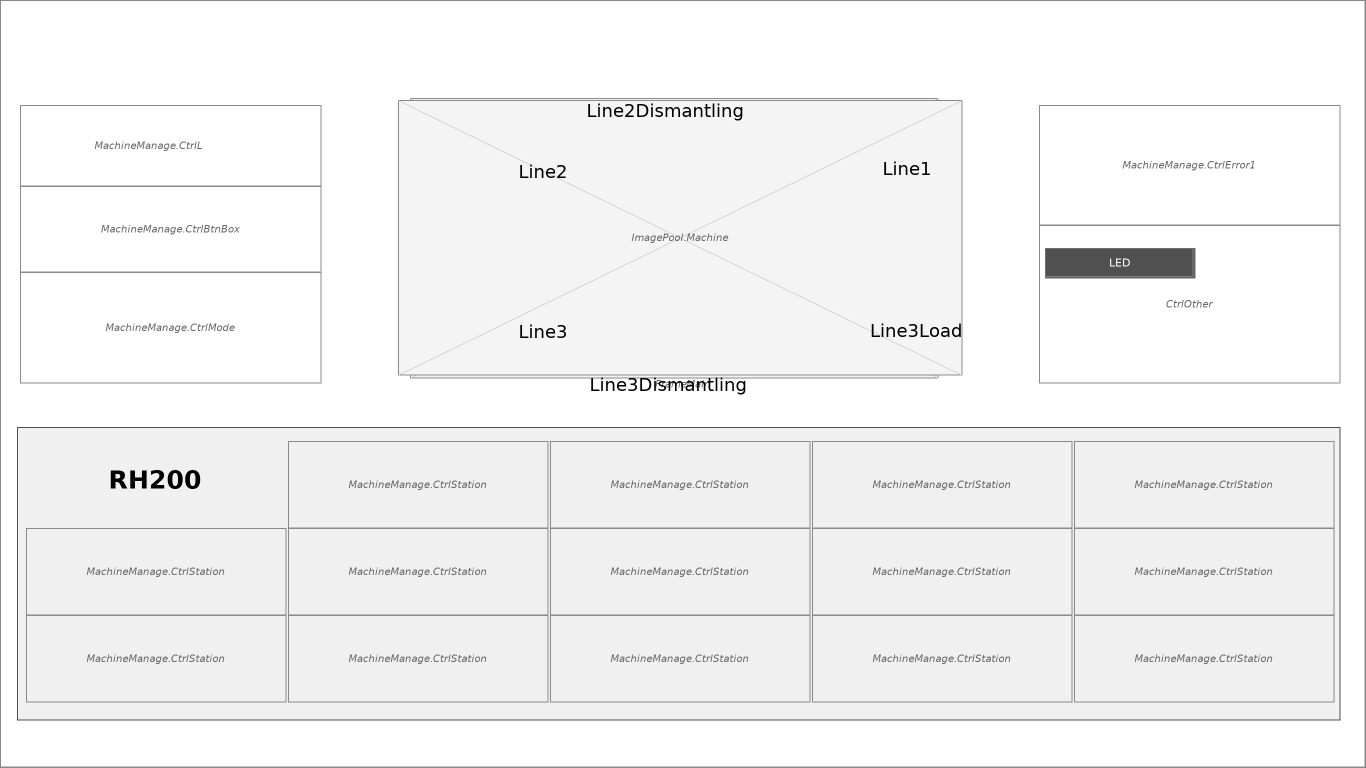
VISUALIZATION PageHome  // 1366x768
    Image (410,98 528x280), image: ImagePool.123
    Frame (0,0 1366x768)
        shows FrameMain()
    Image (398,100 564x275), image: ImagePool.Machine
    Rectangle (17,427 1323x293)
    Frame (20,105 301x81)
        shows MachineManage.CtrlLanguage(System := G_stSystem)
    Frame (20,186 301x86)
        shows MachineManage.CtrlBtnBox(System := G_stSystem)
    Frame (20,272 301x111)
        shows MachineManage.CtrlMode(System := G_stSystem)
    Frame (288,528 260x87)
        shows MachineManage.CtrlStation(System := G_stSystem, Station := G_arrStation[5])
    Frame (550,528 260x87)
        shows MachineManage.CtrlStation(System := G_stSystem, Station := G_arrStation[6])
    Frame (812,528 260x87)
        shows MachineManage.CtrlStation(System := G_stSystem, Station := G_arrStation[7])
    Frame (1074,528 260x87)
        shows MachineManage.CtrlStation(System := G_stSystem, Station := G_arrStation[8])
    Frame (26,615 260x87)
        shows MachineManage.CtrlStation(System := G_stSystem, Station := G_arrStation[9])
    Frame (288,615 260x87)
        shows MachineManage.CtrlStation(System := G_stSystem, Station := G_arrStation[10])
    Frame (550,615 260x87)
        shows MachineManage.CtrlStation(System := G_stSystem, Station := G_arrStation[11])
    Frame (812,615 260x87)
        shows MachineManage.CtrlStation(System := G_stSystem, Station := G_arrStation[12])
    Frame (1074,615 260x87)
        shows MachineManage.CtrlStation(System := G_stSystem, Station := G_arrStation[13])
    Frame (288,441 260x87)
        shows MachineManage.CtrlStation(System := G_stSystem, Station := G_arrStation[0])
    Frame (550,441 260x87)
        shows MachineManage.CtrlStation(System := G_stSystem, Station := G_arrStation[1])
    Frame (812,441 260x87)
        shows MachineManage.CtrlStation(System := G_stSystem, Station := G_arrStation[2])
    Frame (1074,441 260x87)
        shows MachineManage.CtrlStation(System := G_stSystem, Station := G_arrStation[3])
    Frame (26,528 260x87)
        shows MachineManage.CtrlStation(System := G_stSystem, Station := G_arrStation[4])
    Frame (1039,105 301x120)
        shows MachineManage.CtrlError1(System := G_stSystem, Error := G_stError.stNow)
    Frame (1039,225 301x158)
        shows CtrlOther()
    Label (866,154 82x30), "Line1"
    Label (502,157 82x30), "Line2"
    Label (502,317 82x30), "Line3"
    Label (866,316 101x30), "Line3Load"
    Label (583,96 165x30), "Line2Dismantling"
    Label (586,370 165x30), "Line3Dismantling"
    Rectangle (202,126 83x56)
    Rectangle (49,451 212x57), "RH200", text list: 'MachineType', text index: GVL_Data.stRecipe.eMachineType
    Button (1045,248 150x30), "LED"
        toggle GVL.Q.bLED
END_VISUALIZATION

(* stored: Version 1.1.0.1, ProductVersion 3.1.4024.3
   Visu PageHome: Id {6f3cc229-475a-49a0-905f-190a42f85a9f} *)
